{attribute 'GeneratedUsingTerminal: EL2602-0010-0016'}
{attribute addProperty BoxType "EL2602-0010-0016"}
{attribute addProperty Id "StatusAT %I*BOOL1"}
{attribute addProperty CRC "697284909"}
{attribute addProperty Size "1"}
TYPE Inputs_298FB92D EXTENDS InputBase_8311D824 :
STRUCT
	{attribute addProperty Name "Status"}
	Status AT %I* : BOOL;
END_STRUCT
END_TYPE

(* stored: Version 1.2.0.0, ProductVersion 3.1.4024.9
   DUT Inputs_298FB92D: Id {810c4d75-8f61-4f19-ad0e-eff68a69b2a2} *)
